RoboDK station: final_gruppe7.rdk

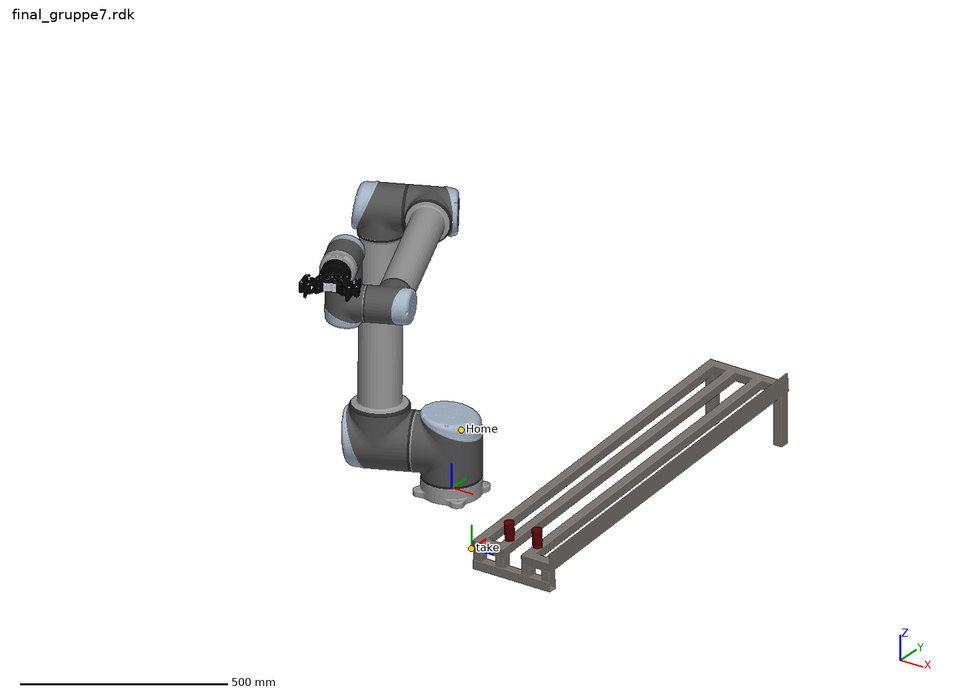
[picture v0: the station drawn from its stored meshes, robots at their saved joint values, targets as dots, program paths as lines]
Station final_gruppe7 (saved by RoboDK 5.5.1). Poses are relative to the parent item; angles as X-Y-Z fixed-axis rotations.
  - frame UR10 Base at (0, 0, 0) mm
    - robot UR10: 6 axes, payload 10 kg, reach 1300 mm, repeatability 0.1 mm, weight 28.9 kg
        modified DH rows (alpha deg, a mm, theta deg, d mm): 0, 0, 0, 118; 90, 0, 180, 0; 0, 612.7, 0, 0; 0, 571.6, 0, 163.9; -90, 0, 0, 115.7; 90, 0, 180, 92.2
        joint limits [-360, -360, -360, -360, -360, -360] to [360, 360, 360, 360, 360, 360]; home [0, -90, -90, 0, 90, 0]; saved at [-65.45, -88.11, -90, 0, 90, 0]
      - tool Gripper RobotiQ 85 Opened, TCP at (0, -20, 130) mm, size 147.4 x 146.8 x 75 mm
  - frame take_plan at (422, -518.71, 162) mm, rotated rx 90 ry 0 rz 90 deg
    - target take (Cartesian target) at (0, 0, 0) mm; joints [270.499, -143.529, -158.107, -98.044, 132.25, -78.379] of UR10
    - target Home (Cartesian target) at (100, 250, -100) mm; joints [72.313, 54.877, -116.065, 61.188, 32.103, 0] of UR10
    - object Magasin_DMH_uten plate at (-160, -210, 110) mm, size 1004.3 x 189.6 x 228 mm, geometry from Magasin_DMH_uten plate.STEP
  - Python program Prog4 (listed below)

--- Python program Prog4 ---
from robodk import *      # RoboDK API
from robolink import *    # Robot toolbox
sim = Robolink()

robot = sim.Item("UR10")
base = sim.Item("UR10 Base")
robot.setPoseFrame(base)
robot_tool = sim.Item("Gripper RobotiQ 85 Opened")
home = sim.Item("Home")
take_plan = sim.Item("take_plan")
take = sim.Item("take")

radios = 53
x = -308
y = -698.71
z = -268

ry_robot = 4.33
ry = 180 - ry_robot

take_plan.setPose(transl(x,y,z) * rotx((-90*pi)/180)* roty((ry*pi)/180)*rotz((180*pi)/180))

robot.setPoseFrame(take_plan)
robot.MoveL(home)
robot.Pause(1000)

robot.MoveL(take.Pose() * transl(radios + 24, radios + 102, -100))
robot.RunInstruction("tfg_grip(10, 80, external_grip=True,stop_if_no_force=False,tool_index=0, blocking=True)", INSTRUCTION_INSERT_CODE)

robot.Pause(1000)

robot.MoveL(take.Pose() * transl(radios + 24, radios + 102, 95))
robot.RunInstruction("tfg_grip(105, 100, external_grip=False,stop_if_no_force=True,tool_index=0, blocking=True)", INSTRUCTION_INSERT_CODE)
robot.Pause(1000)

robot.MoveL(take.Pose() * transl(radios + 24, 250 + radios , 80))
robot.Pause(1000)

robot.MoveL(take.Pose() * transl(radios + 24, 250 + radios , -100))
robot.Pause(1000)
